// TIA Portal V17 export
// export: Created 2025-03-13T10:30:56.3876909Z, ExportSetting WithDefaults, DisplayName Totally Integrated Automation Portal, DisplayVersion V17 Update 8, DisplayName TIA Portal Openness, DisplayVersion V17 Update 8, DisplayName TIA Portal Version Control Interface, DisplayVersion V17, DisplayName SINAMICS Startdrive Advanced, DisplayVersion V17 SP2, DisplayName SINAMICS Startdrive G110M, G120, G120C, G120D, G120P, G115D, DisplayVersion V17 SP2, DisplayName SINAMICS Startdrive G130, G150, S120, S150, SINAMICS MV, S210, DisplayVersion V17 SP2, DisplayName STEP 7 Professional, DisplayVersion V17 Update 8, DisplayName SINUMERIK ONE STEP 7 Toolbox, DisplayVersion V17 Update 12, DisplayName SINUMERIK 840D sl STEP 7 Toolbox, DisplayVersion V17 Update 12, DisplayName STEP 7 Safety, DisplayVersion V17 Update 6, DisplayName WinCC Advanced, DisplayVersion V17 Update 8
DATA_BLOCK "DB1799_ASPIRATION_AUX"   // DB1799
{ S7_Optimized_Access := 'FALSE'; DB_Accessible_From_OPC_UA := 'FALSE' }
VERSION : 0.1
// stored: AutoNumber false, DBAccessibleFromOPCUA false, DBAccessibleFromWebserver true, IsOnlyStoredInLoadMemory false, IsWriteProtectedInAS false
   VAR RETAIN
      UNIT_01_ASPIRATION : Struct
         NORMALIZED_VALUE : Real := 0.5443432;
         SCALED_VALUE : Real := 136.0858;
         LOW_PRESSURE_ALARM : Bool := FALSE;   // ASPIRATION PRESSURE TOO LOW ALARM
         HIGH_PRESSURE_ALARM : Bool := FALSE;   // ASPIRATION PRESSURE TOO HIGH ALARM
         LOW_PRESSURE_WARNING : Bool := FALSE;   // ASPIRATION PRESSURE TOO LOW WARNING
         HIGH_PRESSURE_WARNING : Bool := FALSE;   // ASPIRATION PRESSURE TOO HIGH WARNING
         FINAL_VALUE : Real := -1.360858;
      END_STRUCT;
      UNIT_02_ASPIRATION : Struct
         NORMALIZED_VALUE : Real := 0.6935076;
         SCALED_VALUE : Real := 173.3769;
         LOW_PRESSURE_ALARM : Bool := FALSE;   // ASPIRATION PRESSURE TOO LOW ALARM
         HIGH_PRESSURE_ALARM : Bool := FALSE;   // ASPIRATION PRESSURE TOO HIGH ALARM
         LOW_PRESSURE_WARNING : Bool := FALSE;   // ASPIRATION PRESSURE TOO LOW WARNING
         HIGH_PRESSURE_WARNING : Bool := FALSE;   // ASPIRATION PRESSURE TOO HIGH WARNING
         FINAL_VALUE : Real := -1.733769;
      END_STRUCT;
      HMI : Struct
         U01_HIGH_LIMIT_ALARM_VALUE : Real := -2.2;
         U01_HIGH_LIMIT_WARNING_VALUE : Real := -1.8;
         U01_LOW_LIMIT_ALARM_VALUE : Real := -0.8;
         U01_LOW_LIMIT_WARNING_VALUE : Real := -1.2;
         U01_SWITCH_ON_BUTTON : Bool := FALSE;
         U01_SWITCH_OFF_BUTTON : Bool := FALSE;
         U02_HIGH_LIMIT_ALARM_VALUE : Real := -2.2;
         U02_HIGH_LIMIT_WARNING_VALUE : Real := -1.8;
         U02_LOW_LIMIT_ALARM_VALUE : Real := -1.0;
         U02_LOW_LIMIT_WARNING_VALUE : Real := -1.2;
         U02_SWITCH_ON_BUTTON : Bool := FALSE;
         U02_SWITCH_OFF_BUTTON : Bool := FALSE;
      END_STRUCT;
      TIMERS : Struct
         TIMER_1 : IEC_TIMER;
         TIMER_2 : IEC_TIMER;
         TIMER_3 : IEC_TIMER;
         TIMER_4 : IEC_TIMER;
         TIMER_5 { S7_SetPoint := 'True'} : IEC_TIMER;
         TIMER_6 { S7_SetPoint := 'True'} : IEC_TIMER;
         TIMER_7 { S7_SetPoint := 'True'} : IEC_TIMER;
         TIMER_8 { S7_SetPoint := 'True'} : IEC_TIMER;
      END_STRUCT;
      UNIT_01_PRESSURE_CONTROL : Struct
         STA_3_PRESSURE_CONTROL : Struct
            NORMALIZED_VALUE : Real := 0.0;
            SCALED_VALUE : Real := 0.0;
            FINAL_VALUE : Real := 0.0;
         END_STRUCT;
      END_STRUCT;
      UNIT_02_PRESSURE_CONTROL : Struct
         STA_3_PRESSURE_CONTROL : Struct
            NORMALIZED_VALUE : Real := 0.0;
            SCALED_VALUE : Real := 0.0;
            FINAL_VALUE : Real := 0.0;
         END_STRUCT;
      END_STRUCT;
   END_VAR
BEGIN
   TIMERS.TIMER_1.PT := T#0MS;
   TIMERS.TIMER_1.IN := FALSE;
   TIMERS.TIMER_2.PT := T#0MS;
   TIMERS.TIMER_2.IN := FALSE;
   TIMERS.TIMER_3.PT := T#0MS;
   TIMERS.TIMER_3.IN := FALSE;
   TIMERS.TIMER_4.PT := T#0MS;
   TIMERS.TIMER_4.IN := FALSE;
   TIMERS.TIMER_5.PT := T#0MS;
   TIMERS.TIMER_5.IN := FALSE;
   TIMERS.TIMER_6.PT := T#0MS;
   TIMERS.TIMER_6.IN := FALSE;
   TIMERS.TIMER_7.PT := T#0MS;
   TIMERS.TIMER_7.IN := FALSE;
   TIMERS.TIMER_8.PT := T#0MS;
   TIMERS.TIMER_8.IN := FALSE;
END_DATA_BLOCK
